FUNCTION NextMinorStep : UDINT
VAR_IN_OUT
	StateVar : UDINT;
END_VAR

NextMinorStep := StateVar := StateVar + 1;

END_FUNCTION

(* stored: Version 1.1.0.1, ProductVersion 3.1.4026.18
   POU NextMinorStep: Id {5f107c54-4b01-089b-079e-34e65a415783}, SpecialFunc None *)
